(* CoDeSys 2.3 export: MAIN_FAST.EXP *)

(* POU MAIN_FAST, ST *)
PROGRAM MAIN_FAST
VAR CONSTANT
	FROELING_MODBUS_ADDRESS: USINT := 9;
END_VAR
VAR
	rs232: FB_SetSerial;
	fbFroeling: FB_Froeling;
(*	froeling: ModbusRtuMaster_KL6x22B;
	froelingIn: MB_KL6inData22B;
	froelingOut: MB_KL6outData22B;
	froelingData: INT;
*)
	uiStateCX5000 AT %I*: UINT;
	uiControlCX5000 AT %Q* : UINT;
	iVoltagePhase1 AT %I* : ARRAY [0..9] OF INT;
	iVoltagePhase2 AT %I* : ARRAY [0..9] OF INT;
	iVoltagePhase3 AT %I* : ARRAY [0..9] OF INT;
	uliStartTimeNextLatch AT %I* : ARRAY [0..1] OF UDINT;
	bWcState AT %I* : BOOL;

	fbAnalyseVoltagePhase1 : FB_ANALYSE_VOLTAGE;
	fbAnalyseVoltagePhase2 : FB_ANALYSE_VOLTAGE;
	fbAnalyseVoltagePhase3 : FB_ANALYSE_VOLTAGE;
	fbA28CH1: FB_SYNC_RELAIS;
	fbA28CH2: FB_SYNC_RELAIS;
	fbA29CH1: FB_SYNC_RELAIS;
	fbA29CH2: FB_SYNC_RELAIS;
	fbA30CH1: FB_SYNC_RELAIS;
	fbA30CH2: FB_SYNC_RELAIS;
	fbA31CH1: FB_SYNC_RELAIS;
	fbA31CH2: FB_SYNC_RELAIS;
	fbA32CH1: FB_SYNC_RELAIS;
	fbA32CH2: FB_SYNC_RELAIS;
	fbA20CH1: FB_SYNC_RELAIS;
	fbA20CH2: FB_SYNC_RELAIS;
	fbA21CH1: FB_SYNC_RELAIS;
	fbA21CH2: FB_SYNC_RELAIS;
	fbA23CH1: FB_SYNC_RELAIS;
	fbA23CH2: FB_SYNC_RELAIS;
	fbA24CH1: FB_SYNC_RELAIS;
	fbA24CH2: FB_SYNC_RELAIS;
	fbA25CH1: FB_SYNC_RELAIS;
	fbA25CH2: FB_SYNC_RELAIS;
	fbA26CH1: FB_SYNC_RELAIS;
	fbA26CH2: FB_SYNC_RELAIS;
	fbA38OGCH1: FB_SYNC_RELAIS;
	fbA38OGCH2: FB_SYNC_RELAIS;
	fbA41OGCH1: FB_SYNC_RELAIS;
	fbA41OGCH2: FB_SYNC_RELAIS;
	fbA43OGCH1: FB_SYNC_RELAIS;
	fbA43OGCH2: FB_SYNC_RELAIS;
	fbA44OGCH1: FB_SYNC_RELAIS;
	fbA44OGCH2: FB_SYNC_RELAIS;
	fbA45OGCH1: FB_SYNC_RELAIS;
	fbA45OGCH2: FB_SYNC_RELAIS;
	fbA48OGCH1: FB_SYNC_RELAIS;
	fbA48OGCH2: FB_SYNC_RELAIS;
	fbA49OGCH1: FB_SYNC_RELAIS;
	fbA49OGCH2: FB_SYNC_RELAIS;
	fbA50OGCH1: FB_SYNC_RELAIS;
	fbA50OGCH2: FB_SYNC_RELAIS;
	fbA52OGCH1: FB_SYNC_RELAIS;
	fbA52OGCH2: FB_SYNC_RELAIS;
	fbA53OGCH1: FB_SYNC_RELAIS;
	fbA53OGCH2: FB_SYNC_RELAIS;
	fbA55OGCH1: FB_SYNC_RELAIS;
	fbA55OGCH2: FB_SYNC_RELAIS;
	fbA56OGCH1: FB_SYNC_RELAIS;
	fbA56OGCH2: FB_SYNC_RELAIS;
	fbA57OGCH1: FB_SYNC_RELAIS;
	fbA57OGCH2: FB_SYNC_RELAIS;
	fbA15OGCH1: FB_SYNC_RELAIS;
	fbA15OGCH2: FB_SYNC_RELAIS;
	fbA17OGCH1: FB_SYNC_RELAIS;
	fbA17OGCH2: FB_SYNC_RELAIS;
	fbA18OGCH1: FB_SYNC_RELAIS;
	fbA18OGCH2: FB_SYNC_RELAIS;
	fbA19OGCH1: FB_SYNC_RELAIS;
	fbA19OGCH2: FB_SYNC_RELAIS;
	fbA21OGCH1: FB_SYNC_RELAIS;
	fbA21OGCH2: FB_SYNC_RELAIS;
	fbA23OGCH1: FB_SYNC_RELAIS;
	fbA23OGCH2: FB_SYNC_RELAIS;
	fbA25OGCH1: FB_SYNC_RELAIS;
	fbA25OGCH2: FB_SYNC_RELAIS;
	fbA26OGCH1: FB_SYNC_RELAIS;
	fbA26OGCH2: FB_SYNC_RELAIS;
	fbA33OGCH1: FB_SYNC_RELAIS;
	fbA33OGCH2: FB_SYNC_RELAIS;
	fbA35OGCH1: FB_SYNC_RELAIS;
	fbA35OGCH2: FB_SYNC_RELAIS;
	fbA36OGCH1: FB_SYNC_RELAIS;
	fbA36OGCH2: FB_SYNC_RELAIS;
	fbA78OGCH1: FB_SYNC_RELAIS;
	fbA78OGCH2: FB_SYNC_RELAIS;
	fbA80OGCH1: FB_SYNC_RELAIS;
	fbA80OGCH2: FB_SYNC_RELAIS;

	lrFrequencyPhase1: LREAL;
	lrFrequencyPhase2: LREAL;
	lrFrequencyPhase3: LREAL;
	bErrorL1: BOOL;
	bErrorL2: BOOL;
	bErrorL3: BOOL;

	bRelayPLC:BOOL;
END_VAR
(*
froeling.UnitID := 10;
froeling.Quantity := 1;
froeling.MBAddr := 30022;
froeling.cbLength := SIZEOF(froelingData);
froeling.pMemoryAddr := ADR(froelingData);
froeling.Timeout := t#8s;
froeling.Execute := TRUE;
*)

fbFroeling(
	modbusSlaveAddress := FROELING_MODBUS_ADDRESS,
	timeout := t#1s,
);

(* Spannungsanalyse *)
fbAnalyseVoltagePhase1(
	uliStartTimeNextLatch := uliStartTimeNextLatch,
	bWcState := bWcState,
	iVoltage := iVoltagePhase1,
	lrFrequency => lrFrequencyPhase1,
	bError => bErrorL1);

fbAnalyseVoltagePhase2(
	uliStartTimeNextLatch := uliStartTimeNextLatch,
	bWcState := bWcState,
	iVoltage := iVoltagePhase2,
	lrFrequency => lrFrequencyPhase2,
	bError => bErrorL2);

fbAnalyseVoltagePhase3(
	uliStartTimeNextLatch := uliStartTimeNextLatch,
	bWcState := bWcState,
	iVoltage := iVoltagePhase3,
	lrFrequency => lrFrequencyPhase3,
	bError => bErrorL3);

(* Relais *)
fbA28CH1(bValue:= , udiDelayNanoSek:= 5800000, tNextZeroVoltage:= fbAnalyseVoltagePhase1.tNextZeroVoltage);
fbA28CH2(bValue:= , udiDelayNanoSek:= 6600000, tNextZeroVoltage:= fbAnalyseVoltagePhase1.tNextZeroVoltage);
fbA29CH1(bValue:= , udiDelayNanoSek:= 6300000, tNextZeroVoltage:= fbAnalyseVoltagePhase1.tNextZeroVoltage);
fbA29CH2(bValue:= , udiDelayNanoSek:= 6500000, tNextZeroVoltage:= fbAnalyseVoltagePhase1.tNextZeroVoltage);
fbA30CH1(bValue:= , udiDelayNanoSek:= 6500000, tNextZeroVoltage:= fbAnalyseVoltagePhase1.tNextZeroVoltage);
fbA30CH2(bValue:= , udiDelayNanoSek:= 5700000, tNextZeroVoltage:= fbAnalyseVoltagePhase1.tNextZeroVoltage);
fbA31CH1(bValue:= , udiDelayNanoSek:= 5700000, tNextZeroVoltage:= fbAnalyseVoltagePhase1.tNextZeroVoltage);
fbA31CH2(bValue:= , udiDelayNanoSek:= 5700000, tNextZeroVoltage:= fbAnalyseVoltagePhase1.tNextZeroVoltage);
fbA32CH1(bValue:= , udiDelayNanoSek:= 6000000, tNextZeroVoltage:= fbAnalyseVoltagePhase2.tNextZeroVoltage);
fbA32CH2(bValue:= , udiDelayNanoSek:= 6000000, tNextZeroVoltage:= fbAnalyseVoltagePhase2.tNextZeroVoltage);
fbA20CH1(bValue:=MAIN.kgGangLampe.Q, udiDelayNanoSek:= 6700000, tNextZeroVoltage:= fbAnalyseVoltagePhase1.tNextZeroVoltage);
fbA20CH2(bValue:=MAIN.kgEgLampe.Q, udiDelayNanoSek:= 5800000, tNextZeroVoltage:= fbAnalyseVoltagePhase1.tNextZeroVoltage);
fbA21CH1(bValue:=MAIN.lagerLampe.Q, udiDelayNanoSek:= 6400000, tNextZeroVoltage:= fbAnalyseVoltagePhase1.tNextZeroVoltage);
fbA21CH2(bValue:= , udiDelayNanoSek:= 6500000, tNextZeroVoltage:= fbAnalyseVoltagePhase1.tNextZeroVoltage);
fbA23CH1(bValue:=MAIN.heizenLampe.Q, udiDelayNanoSek:= 6500000, tNextZeroVoltage:= fbAnalyseVoltagePhase2.tNextZeroVoltage);
fbA23CH2(bValue:=MAIN.waschenLampeS.Q, udiDelayNanoSek:= 6300000, tNextZeroVoltage:= fbAnalyseVoltagePhase2.tNextZeroVoltage);
fbA24CH1(bValue:=MAIN.waschenLampeNM.Q, udiDelayNanoSek:= 6300000, tNextZeroVoltage:= fbAnalyseVoltagePhase2.tNextZeroVoltage);
fbA24CH2(bValue:=MAIN.hobbyLampeN.Q, udiDelayNanoSek:= 6000000, tNextZeroVoltage:= fbAnalyseVoltagePhase2.tNextZeroVoltage);
fbA25CH1(bValue:=MAIN.vorratLampe.Q, udiDelayNanoSek:= 6000000, tNextZeroVoltage:= fbAnalyseVoltagePhase2.tNextZeroVoltage);
fbA25CH2(bValue:=MAIN.hobbyLampeS.Q, udiDelayNanoSek:= 6300000, tNextZeroVoltage:= fbAnalyseVoltagePhase2.tNextZeroVoltage);
fbA26CH1(bValue:= , udiDelayNanoSek:= 6300000, tNextZeroVoltage:= fbAnalyseVoltagePhase2.tNextZeroVoltage);
fbA26CH2(bValue:= , udiDelayNanoSek:= 6150000, tNextZeroVoltage:= fbAnalyseVoltagePhase2.tNextZeroVoltage);
fbA38OGCH1(bValue:= , udiDelayNanoSek:= 6000000, tNextZeroVoltage:= fbAnalyseVoltagePhase1.tNextZeroVoltage);
fbA38OGCH2(bValue:= , udiDelayNanoSek:= 6200000, tNextZeroVoltage:= fbAnalyseVoltagePhase1.tNextZeroVoltage);
fbA41OGCH1(bValue:= , udiDelayNanoSek:= 6200000, tNextZeroVoltage:= fbAnalyseVoltagePhase2.tNextZeroVoltage);
fbA41OGCH2(bValue:=MAIN.ogBadLampeOM.Q, udiDelayNanoSek:= 5600000, tNextZeroVoltage:= fbAnalyseVoltagePhase2.tNextZeroVoltage);
fbA43OGCH1(bValue:= , udiDelayNanoSek:= 5800000, tNextZeroVoltage:= fbAnalyseVoltagePhase1.tNextZeroVoltage);
fbA43OGCH2(bValue:= , udiDelayNanoSek:= 5800000, tNextZeroVoltage:= fbAnalyseVoltagePhase1.tNextZeroVoltage);
fbA44OGCH1(bValue:=MAIN.ogKindLampeN.Q, udiDelayNanoSek:= 5800000, tNextZeroVoltage:= fbAnalyseVoltagePhase1.tNextZeroVoltage);
fbA44OGCH2(bValue:=MAIN.ogKindLampeS.Q, udiDelayNanoSek:= 5800000, tNextZeroVoltage:= fbAnalyseVoltagePhase1.tNextZeroVoltage);
fbA45OGCH1(bValue:=MAIN.ogKindLampeM.Q, udiDelayNanoSek:= 5800000, tNextZeroVoltage:= fbAnalyseVoltagePhase1.tNextZeroVoltage);
fbA45OGCH2(bValue:=MAIN.dgKindLampe.Q, udiDelayNanoSek:= 5800000, tNextZeroVoltage:= fbAnalyseVoltagePhase1.tNextZeroVoltage);
fbA48OGCH1(bValue:= , udiDelayNanoSek:= 6000000, tNextZeroVoltage:= fbAnalyseVoltagePhase2.tNextZeroVoltage);
fbA48OGCH2(bValue:= , udiDelayNanoSek:= 6000000, tNextZeroVoltage:= fbAnalyseVoltagePhase2.tNextZeroVoltage);
fbA49OGCH1(bValue:= , udiDelayNanoSek:= 6000000, tNextZeroVoltage:= fbAnalyseVoltagePhase2.tNextZeroVoltage);
fbA49OGCH2(bValue:= , udiDelayNanoSek:= 5800000, tNextZeroVoltage:= fbAnalyseVoltagePhase2.tNextZeroVoltage);
fbA50OGCH1(bValue:= , udiDelayNanoSek:= 6000000, tNextZeroVoltage:= fbAnalyseVoltagePhase2.tNextZeroVoltage);
fbA50OGCH2(bValue:= , udiDelayNanoSek:= 5600000, tNextZeroVoltage:= fbAnalyseVoltagePhase2.tNextZeroVoltage);
fbA52OGCH1(bValue:= , udiDelayNanoSek:= 6000000, tNextZeroVoltage:= fbAnalyseVoltagePhase2.tNextZeroVoltage);
fbA52OGCH2(bValue:= , udiDelayNanoSek:= 6000000, tNextZeroVoltage:= fbAnalyseVoltagePhase2.tNextZeroVoltage);
fbA53OGCH1(bValue:= , udiDelayNanoSek:= 5900000, tNextZeroVoltage:= fbAnalyseVoltagePhase2.tNextZeroVoltage);
fbA53OGCH2(bValue:= , udiDelayNanoSek:= 5900000, tNextZeroVoltage:= fbAnalyseVoltagePhase2.tNextZeroVoltage);
fbA55OGCH1(bValue:= , udiDelayNanoSek:= 5900000, tNextZeroVoltage:= fbAnalyseVoltagePhase3.tNextZeroVoltage);
fbA55OGCH2(bValue:= , udiDelayNanoSek:= 5600000, tNextZeroVoltage:= fbAnalyseVoltagePhase3.tNextZeroVoltage);
fbA56OGCH1(bValue:= , udiDelayNanoSek:= 5600000, tNextZeroVoltage:= fbAnalyseVoltagePhase3.tNextZeroVoltage);
fbA56OGCH2(bValue:= , udiDelayNanoSek:= 5700000, tNextZeroVoltage:= fbAnalyseVoltagePhase3.tNextZeroVoltage);
fbA57OGCH1(bValue:= , udiDelayNanoSek:= 5600000, tNextZeroVoltage:= fbAnalyseVoltagePhase3.tNextZeroVoltage);
fbA57OGCH2(bValue:= , udiDelayNanoSek:= 5900000, tNextZeroVoltage:= fbAnalyseVoltagePhase3.tNextZeroVoltage);

fbA15OGCH1(bValue:=MAIN.essenLampeNW.Q, udiDelayNanoSek:= 6100000, tNextZeroVoltage:= fbAnalyseVoltagePhase1.tNextZeroVoltage);
fbA15OGCH2(bValue:= , udiDelayNanoSek:= 6300000, tNextZeroVoltage:= fbAnalyseVoltagePhase1.tNextZeroVoltage);
fbA17OGCH1(bValue:=MAIN.schlafenLampeO.Q, udiDelayNanoSek:= 6100000, tNextZeroVoltage:= fbAnalyseVoltagePhase2.tNextZeroVoltage);
fbA17OGCH2(bValue:= , udiDelayNanoSek:= 6100000, tNextZeroVoltage:= fbAnalyseVoltagePhase2.tNextZeroVoltage);
fbA18OGCH1(bValue:=MAIN.wohnenLampeSW.Q, udiDelayNanoSek:= 6100000, tNextZeroVoltage:= fbAnalyseVoltagePhase2.tNextZeroVoltage);
fbA18OGCH2(bValue:= , udiDelayNanoSek:= 6100000, tNextZeroVoltage:= fbAnalyseVoltagePhase2.tNextZeroVoltage);
fbA19OGCH1(bValue:= , udiDelayNanoSek:= 6100000, tNextZeroVoltage:= fbAnalyseVoltagePhase2.tNextZeroVoltage);
fbA19OGCH2(bValue:= , udiDelayNanoSek:= 6100000, tNextZeroVoltage:= fbAnalyseVoltagePhase2.tNextZeroVoltage);
fbA21OGCH1(bValue:= , udiDelayNanoSek:= 6000000, tNextZeroVoltage:= fbAnalyseVoltagePhase3.tNextZeroVoltage);
fbA21OGCH2(bValue:= , udiDelayNanoSek:= 6100000, tNextZeroVoltage:= fbAnalyseVoltagePhase3.tNextZeroVoltage);
fbA23OGCH1(bValue:= , udiDelayNanoSek:= 6100000, tNextZeroVoltage:= fbAnalyseVoltagePhase2.tNextZeroVoltage);
fbA23OGCH2(bValue:= , udiDelayNanoSek:= 6100000, tNextZeroVoltage:= fbAnalyseVoltagePhase2.tNextZeroVoltage);
fbA25OGCH1(bValue:=MAIN.kochenLampeO.Q, udiDelayNanoSek:= 6100000, tNextZeroVoltage:= fbAnalyseVoltagePhase2.tNextZeroVoltage);
fbA25OGCH2(bValue:=MAIN.kochenLampeN.Q, udiDelayNanoSek:= 6100000, tNextZeroVoltage:= fbAnalyseVoltagePhase2.tNextZeroVoltage);
fbA26OGCH1(bValue:=MAIN.speisLampe.Q , udiDelayNanoSek:= 6100000, tNextZeroVoltage:= fbAnalyseVoltagePhase2.tNextZeroVoltage);
fbA26OGCH2(bValue:= , udiDelayNanoSek:= 6100000, tNextZeroVoltage:= fbAnalyseVoltagePhase2.tNextZeroVoltage);
fbA33OGCH1(bValue:=MAIN.egBadLampeON.Q, udiDelayNanoSek:= 6100000, tNextZeroVoltage:= fbAnalyseVoltagePhase1.tNextZeroVoltage);
fbA33OGCH2(bValue:= , udiDelayNanoSek:= 6100000, tNextZeroVoltage:= fbAnalyseVoltagePhase1.tNextZeroVoltage);
fbA35OGCH1(bValue:=MAIN.arbeitenLampeN.Q, udiDelayNanoSek:= 6300000, tNextZeroVoltage:= fbAnalyseVoltagePhase3.tNextZeroVoltage);
fbA35OGCH2(bValue:=MAIN.arbeitenLampeS.Q, udiDelayNanoSek:= 6200000, tNextZeroVoltage:= fbAnalyseVoltagePhase3.tNextZeroVoltage);
fbA36OGCH1(bValue:=MAIN.arbeitenLampeSW.Q, udiDelayNanoSek:= 6400000, tNextZeroVoltage:= fbAnalyseVoltagePhase3.tNextZeroVoltage);
fbA36OGCH2(bValue:= , udiDelayNanoSek:= 6300000, tNextZeroVoltage:= fbAnalyseVoltagePhase3.tNextZeroVoltage);
fbA78OGCH1(bValue:= , udiDelayNanoSek:= 5800000, tNextZeroVoltage:= fbAnalyseVoltagePhase3.tNextZeroVoltage);
fbA78OGCH2(bValue:=MAIN.dachbodenLampe.Q, udiDelayNanoSek:= 5800000, tNextZeroVoltage:= fbAnalyseVoltagePhase3.tNextZeroVoltage);
fbA80OGCH1(bValue:= , udiDelayNanoSek:= 5500000, tNextZeroVoltage:= fbAnalyseVoltagePhase1.tNextZeroVoltage);
fbA80OGCH2(bValue:= , udiDelayNanoSek:= 5500000, tNextZeroVoltage:= fbAnalyseVoltagePhase1.tNextZeroVoltage);
END_PROGRAM
